FUNCTION_BLOCK ILOCK_SR (* Realizes a chainable momentary latch with interlock (BOOL interface) *)
  (* Standard: 61499-1; Description: Copyright (c) 2026 Meisterschulen am Ostbahnhof *)
  (* Version 1.0, 2026-05-07, Gemini CLI, Meisterschulen am Ostbahnhof, initial version *)
  PACKAGE logiBUS::signalprocessing::interlock;
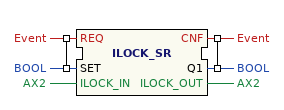
  EVENT_INPUT
    REQ WITH SET; (* Execution Request *)
  END_EVENT
  EVENT_OUTPUT
    CNF WITH Q1; (* Execution Confirmation *)
  END_EVENT
  VAR_INPUT
    SET : BOOL; (* Momentary Set signal *)
  END_VAR
  VAR_OUTPUT
    Q1 : BOOL; (* Output *)
  END_VAR
  SOCKETS
    ILOCK_IN : adapter::types::bidirectional::AX2;
  END_SOCKETS
  PLUGS
    ILOCK_OUT : adapter::types::bidirectional::AX2;
  END_PLUGS
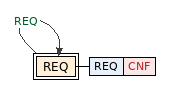
  EC_STATES
    REQ : REQ -> CNF;
  END_STATES
  EC_TRANSITIONS
    REQ TO REQ := REQ;
  END_TRANSITIONS
  ALGORITHM REQ IN ST:
(* Momentary latch: Q1 is active if SET is active AND no other element is set *)
Q1 := SET AND NOT (ILOCK_IN.DO1 OR ILOCK_OUT.DI1);

(* Propagate status *)
ILOCK_IN.DI1 := Q1;
ILOCK_OUT.DO1 := Q1;
  END_ALGORITHM
END_FUNCTION_BLOCK
